// TIA Portal project "babu_pulsesPositiveNegative" (V15)

(* hardware
DEVICE "S7-1200 station_1"  S7-1200 Station
   slot 0: "Rack_0"  S7-1200 Rack  Rack  V1.0
   slot 1: "PLC_1"  CPU 1212C DC/DC/DC  6ES7 212-1AE40-0XB0  V4.2
*)

// ===== PLC "PLC_1"  CPU 1212C DC/DC/DC =====

VAR_GLOBAL   // PLC tag table "Default tag table"
   "IP MEM" AT %M0.0 : Bool;
   "IP" AT %M0.1 : Bool;
   "MEM 2" AT %M0.2 : Bool;
   "OP 2" AT %Q0.0 : Bool;
   "OP 2 MEM" AT %M0.3 : Bool;
   "IP2" AT %M0.4 : Bool;
   "IP3" AT %M0.5 : Bool;
   "OP3" AT %M0.6 : Bool;
   "MEM31" AT %M0.7 : Bool;
   "OP31" AT %M1.0 : Bool;
   "ST3" AT %M1.1 : Bool;
END_VAR

// folder: System blocks/Program resources

DATA_BLOCK "IEC_Timer_0_DB"   // DB1
{ S7_Optimized_Access := 'TRUE' }
AUTHOR : Simatic
FAMILY : IEC
NAME : IEC_TMR
VERSION : 1.0
// stored: InstanceOfName IEC_TIMER
"IEC_TIMER"
BEGIN
END_DATA_BLOCK

// folder: (top level)

ORGANIZATION_BLOCK "Main"   // OB1, LAD, ProgramCycle
TITLE = "Main Program Sweep (Cycle)"
{ S7_Optimized_Access := 'TRUE' }
VERSION : 0.1
   VAR_INPUT
      Initial_Call : Bool;   // Initial call of this OB
      Remanence : Bool;   // =True, if remanent data are available
   END_VAR
   VAR_TEMP   // added for the SCL form of the ladder/FBD networks
      _w1 : Bool;
   END_VAR
BEGIN

REGION Network 1
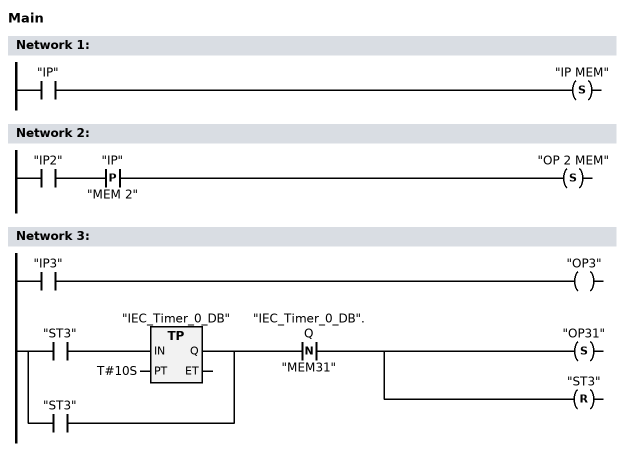
   RUNG wire#powerrail
      Contact( "IP" )
      S_Coil( "IP MEM" )
   END_RUNG
   // the same network as SCL:
   IF "IP" THEN "IP MEM" := TRUE; END_IF;
END_REGION

REGION Network 2
   RUNG wire#powerrail
      Contact( "IP2" )
      P_Contact(operand := "IP", bit := "MEM 2")
      S_Coil( "OP 2 MEM" )
   END_RUNG
   // the same network as SCL:
   #_w1 := "IP2" AND "IP" AND NOT "MEM 2";   // rising edge of "IP"
   "MEM 2" := "IP";
   IF #_w1 THEN "OP 2 MEM" := TRUE; END_IF;
END_REGION

REGION Network 3
   "OP3" := "IP3";
   "IEC_Timer_0_DB".TP(IN := "ST3", PT := T#10S);
   #_w1 := ("IEC_Timer_0_DB".Q OR "ST3") AND NOT "IEC_Timer_0_DB".Q AND "MEM31";   // falling edge of "IEC_Timer_0_DB".Q
   "MEM31" := "IEC_Timer_0_DB".Q;
   IF #_w1 THEN
       "OP31" := TRUE;
       "ST3" := FALSE;
   END_IF;
END_REGION
END_ORGANIZATION_BLOCK